ABB RAPID module: 0005A12C

MODULE Module1
    CONST robtarget Target_CenterSheet:=[[148.5,105,30],[0,1,0,0],[0,0,0,0],[9E+09,9E+09,9E+09,9E+09,9E+09,9E+09]];
ENDMODULE
